// TIA Portal V18 export
VAR_GLOBAL   // PLC tag table "Default tag table"
   "Motor start" AT %I0.0 : Bool;
   "Motor Stop" AT %I0.1 : Bool;
   Tag_2 AT %I0.2 : Bool;
   Tag_4 AT %I0.3 : Bool;
   "Motor running LED" AT %Q0.0 : Bool;
   "Motor contactor" AT %Q0.2 : Bool;
   Tag_1 AT %M10.0 : Bool;
   Tag_3 AT %M10.1 : Bool;
   System_Byte AT %MB88 : Byte;
   FirstScan AT %M88.0 : Bool;
   DiagStatusUpdate AT %M88.1 : Bool;
   AlwaysTRUE AT %M88.2 : Bool;
   AlwaysFALSE AT %M88.3 : Bool;
   "System_Byte(1)" AT %MB88 : Byte;
   Clock_Byte AT %MB0 : Byte;
   Clock_10Hz AT %M0.0 : Bool;
   Clock_5Hz AT %M0.1 : Bool;
   "Clock_2.5Hz" AT %M0.2 : Bool;
   Clock_2Hz AT %M0.3 : Bool;
   "Clock_1.25Hz" AT %M0.4 : Bool;
   Clock_1Hz AT %M0.5 : Bool;
   "Clock_0.625Hz" AT %M0.6 : Bool;
   "Clock_0.5Hz" AT %M0.7 : Bool;
   Alarm AT %MW40 : Word;
   Tag_5 AT %M40.0 : Bool;
END_VAR
